TYPE TComplexStruct :
STRUCT
	intVal : INT:=1200;
	dintArr: ARRAY[0..3] OF DINT:=[ 1,2,3,4];
	boolVal: BOOL := FALSE;
	byteVal: BYTE:=10;
	stringVal : STRING(5) := 'hallo';
	simpleStruct1: TSimpleStruct;
END_STRUCT
END_TYPE

(* stored: Version 1.1.0.1, ProductVersion 3.1.4022.18
   DUT TComplexStruct: Id {100425cf-15b8-4438-b402-de0773c8381f} *)
